FUNCTION_BLOCK FB_MovingAverageLReal
VAR_INPUT
	ValueToAdd : LREAL;
END_VAR
VAR_IN_OUT
	AverageArray  : ARRAY [*] OF LREAL;
END_VAR
VAR_OUTPUT
	CurrentValue : LREAL;
END_VAR
VAR
	CurrentIndex : UINT;
END_VAR
VAR_TEMP
	I: DINT;
	Sum: LREAL;
	ArrayLength : UINT;
END_VAR

// Compute average over array.
// The order of this addition and MOD are important to avoid going out of bounds.
ArrayLength := TO_UINT(UPPER_BOUND(AverageArray, 1) - LOWER_BOUND(AverageArray, 1) + 1);
AverageArray[CurrentIndex] := ValueToAdd;
CurrentIndex := CurrentIndex + 1;
CurrentIndex := CurrentIndex MOD ArrayLength;
FOR I := LOWER_BOUND(AverageArray, 1) TO UPPER_BOUND(AverageArray, 1) BY 1 DO
	Sum := Sum + AverageArray[I];
END_FOR
CurrentValue := Sum / ArrayLength;

END_FUNCTION_BLOCK

(* stored: Version 1.1.0.1, ProductVersion 3.1.4022.16
   POU FB_MovingAverageLReal: Id {f20306fc-a20b-432e-8480-9fba39ec7c43}, SpecialFunc None *)
